(* IEC 61131-3 sources: uPC2_EMCTEST/UPC2_EMCTEST/UPC2_EMCTEST/Source/Definitions, 5 files *)

(* ---- UserDefinedDataType.st.st ---- *)
(*----------------------------------
         ADD HERE YOUR TYPES!
----------------------------------*)
TYPE
    (**STone project GIUD*)
    StonePrjGUID:
        STRUCT
            Grp1 : STRING[8];
            Grp2 : STRING[4];
            Grp3 : STRING[4];
            Grp4 : STRING[4];
            Grp5 : STRING[12];
        END_STRUCT;

    (**Date position range*)
    DatePosRange : UINT(0..99);

    (**Time Struct used to change RTC*)
    TimeRTC: STRUCT
        (**Hourh*)  {ATTRIBUTE UOM HOUR}
        Hour        : UINT(0..23);
        (**Minute*) {ATTRIBUTE UOM MINUTE}
        Minute      : UINT(0..59);
        (**Second*){ATTRIBUTE UOM SECOND}
        Second      : UINT(0..59);
        (**Millisecond*){ATTRIBUTE UOM MILLISECOND}
        Millisecond : UINT(0..999);
    END_STRUCT;

    (**Date Struct used to change RTC*)
    DateRTC: STRUCT
        (**Day*)    {ATTRIBUTE UOM DAY}
        Day         : UINT(1..31);
        (**Month*)  {ATTRIBUTE UOM MONTH}
        Month       : UINT(1..12);
        (**Year*)   {ATTRIBUTE UOM YEAR}
        Year        : UINT(2021..2200);
    END_STRUCT;

    (**Date and time Struct used to change RTC*)
    DateTimeRTC: STRUCT
        (**Day*)    {ATTRIBUTE UOM DAY}
        Day         : UINT(1..31);
        (**Month*)  {ATTRIBUTE UOM MONTH}
        Month       : UINT(1..12);
        (**Year*)   {ATTRIBUTE UOM YEAR}
        Year        : UINT(2021..2200);
        (**Hourh*)  {ATTRIBUTE UOM HOUR}
        Hour        : UINT(0..23);
        (**Minute*) {ATTRIBUTE UOM MINUTE}
        Minute      : UINT(0..59);
        (**Second*){ATTRIBUTE UOM SECOND}
        Second      : UINT(0..59);
        (**Millisecond*){ATTRIBUTE UOM MILLISECOND}
        Millisecond : UINT(0..999);
    END_STRUCT;

    (**Units measure zone*)
    UOM_ZONE :
        (
        (**No Zone*)
        NONE,
        (**International System Zone [°C/bar]*)
        SI,
        (**Imperial Zone [°F/psi]*)
        Imperial
        );

   (**Unit status type*)
    UNIT_STATUS:
    (
        NOT_Used,                   (**Bacnet compatibility*)
        UnitON,                     (**Unit ON*)
        OffByAlarm,                 (**Off By Alarm*)
        OffByBMS,                   (**Off By BMS*)
        OffByScheduler,             (**Off By Scheduler*)
        OffByDI,                    (**Off By Digital Input*)
        OffByKeyboard,              (**Off By Keyboard*)
        OffByNetwork,               (**Off By Network*)
        Manual,                     (**Unit manual mode active*)
        ChangeOver,                 (**ChangeOver*)
        SwitchON,                   (**Switch ON*)
        ShutDown,                   (**Shut Down*)
        PreConditioning,            (**Pre-Conditioning*)
        Dehumidification,           (**Dehumidification*)
        Antifreeze,                 (**Antifreeze*)
        Defrost,                    (**Defrost*)
        AirPressure_Flow,           (**Air Pressure/Flow*)
        AirQuality,                 (**Air Quality*)
        Cooling,                    (**Cooling*)
        Heating,                    (**Heating*)
        FreeCooling,                (**FreeCooling*)
        FreeHeating,                (**FreeHeating*)
        LowTemperatureControl,      (**Low Temperature Control*)
        HighTemperatureControl,     (**High Temperature Control*)
        TestIO,                     (**Test I/O*)
        DHW,                        (**Domestic Hot Water*)
        InactivityStart,            (**Inactivity Start*)
        HighSaturationHumidity,     (**High Saturation Humidity*)
        Purging                     (**Purging*)
    );

    (**List of Quick Menu position*)
    QUICK_MENU:
    (
        (**Selected Loop OnOff*)
        OnOff,
        (**Selcted Loop Set*)
        Set,
        (**Selected Loop Info*)
        Info
    );

    (**Current state of HMI - Used to manage LogoMask/LanguageMask/MainMask transition*)
    State_HMI:
    (
        Wait,
        DisplayLogoMask,
        DisplayLanguageMask,
        DisplayMainMask
    );

    (**Serial port configuration (Parity and Stop bits)*)
    Serial_ParityStopBits :
    (
        (**NONE-1*)
        NONE_1,
        (**NONE-2*)
        NONE_2,
        (**EVEN-1*)
        EVEN_1,
        (**EVEN-2*)
        EVEN_2,
        (**ODD-1*)
        ODD_1,
        (**ODD-2*)
        ODD_2
    );

    (**Serial port baud rate configuration*)
    Serial_Speed :
    (
        (**Baud rate 1200*)
        Baud_1200,
        (**Baud rate 2400*)
        Baud_2400,
        (**Baud rate 4800*)
        Baud_4800,
        (**Baud rate 9600*)
        Baud_9600,
        (**Baud rate 19200*)
        Baud_19200,
        (**Baud rate 38400*)
        Baud_38400,
        (**Baud rate 57600*)
        Baud_57600,
        (**Baud rate 115200*)
        Baud_115200,
        (**Baud rate 375000*)
        Baud_375000
    );

    (**Type of password used for Login procedure*)
    LOGIN_PASSWORD :
    (
        User,
        Service,
        Manufacturer,
        System
    );

    (**Used by APPLICA to manage clock and timezone*)
    APPsConfigRTC:
        STRUCT
        	(**Every time it's value change the PLC change it's RTC*)
        	SetRTC     : BOOL;
            (**New "Date and Time" used to update the RTC*)
        	DateTime   : DATE_AND_TIME;
        	(**New "Time Zone" used to update the RTC*)
        	TimeZone   : STRING;
        END_STRUCT;

END_TYPE

(* ---- VAR_GLOBAL.st ---- *)
USING System;
USING System.Timer;
(*----------------------------------
         ADD HERE YOUR VARS!
----------------------------------*)
VAR_GLOBAL
    (**Restore application to defualt settings (FALSE=Disabled, TRUE=Enabled)*)
	Restoredefault   : BOOL;
    (**Instance to manage comunication between Client&Salve in Modbus client protocol with Fieldbus port*)
//    ClientModbus_pCO : MBM_Template_pCO;

    {REGION SYSTEM INFO}
        (**Retain writings number*)
        RetainWrN       : UDINT;
        (**Task Main live counter*)
        TaskMainLiveCnt : UINT;
        (**Task Main execution time*)
        {ATTRIBUTE UOM MILLISECOND}
        TaskMainExeT    : UDINT;
        (**Current System Time*)
        {ATTRIBUTE UOM MILLISECOND}
        CurrSysT        : UDINT;
        (**Task Main current execution time*)
        {ATTRIBUTE UOM MILLISECOND}
        TaskMainCurrT   : UDINT;

        (**System Info structure*)
        SysInfo         : SystemInfo;
        (**Hardware Info structure*)
        HardwareInfo    : HardwareDescription;
        (**Prject information*)
        InfoProject     : ProjectInfo;
        (**Product information read in OTP memory*)
        InfoProduct     : ProductInfo;

        (**PLC SW can GO*)
        Go_PLC          : BOOL;

        (**Device model*)
		DeviceType      : UINT;
        (**Board type*)
        BoardType       : UINT;
        (**Target machine type*)
		MachineType     : UINT;
        (**Target hardware code*)
		HwCode          : UINT;

        RetainMemWrites : ULINT;

        (**Stone project GUID*)
        GUID : StonePrjGUID;
    {ENDREGION}

    {REGION Used by APPLICA to manage clock and timeZONE}
        APPsCfgRTC : APPsConfigRTC;
    {ENDREGION}

    {REGION HMI}
        (**Logged in pGD1 display as Service*)
    	Access_Service : BOOL;
        (**Logged in pGD1 display as User*)
    	Access_User    : BOOL;
        (**Logged in pGD1 display as Manufacturer*)
    	Access_Manuf   : BOOL;
        (**Logged in pGD1 display as System Manager*)
    	Access_Sys     : BOOL;
        (**Switch to TRUE or FALSE every second*)
        Blink          : BOOL;
        (**Password used for Loging procedure (User, Service, Manufacturer, System)*) {METADATA MIN_VAL 0} {METADATA MAX_VAL 3}
        LoginPwdType   : USINT;

    	{REGION Management of "Date and Hour" displayed by pGD1 display}
            (**Current local time (read only)*)
            CurrLocTime    : DateTimeRTC;
            (**UTC Date and Time*)
            TimeUTC        : DATE_AND_TIME;
            (**Local Date and Time based on current time zone*)
            LocDateAndTime : DATE_AND_TIME;
            (**Local time based on current time zone*)
            LocTime        : DateTime;
            (**Current day of week*)
            Day_Week       : DayOfWeek(0..6);
            (**Set clock settings by Net*)
            SetClockByNet  : BOOL;
        {ENDREGION}

        {REGION Date and time changing management by Network}
            (**Values of Date and Time used to modify RTC by network*)
            NewDateTimeByNet  : DateTimeRTC;
        {ENDREGION}

        {REGION Date and time changing management by pGD1}
            (**Values of Date and Time used to modify clock by pGD1*)
            DateTimeBypGD1 : TimeRTC;

            (**Date element position P1, the date format is P1/P2/P3*) {METADATA MIN_VAL DateP1Lmin} {METADATA MAX_VAL DateP1Lmax}
            DateP1     : DatePosRange;
            (**Date element position P1 limit min*)
            DateP1Lmin : DatePosRange;
            (**Date element position P1 limit max*)
            DateP1Lmax : DatePosRange;

            (**Date element position P2, the date format is P1/P2/P3*) {METADATA MIN_VAL DateP2Lmin} {METADATA MAX_VAL DateP2Lmax}
            DateP2     : DatePosRange;
            (**Date element position P2 limit min*)
            DateP2Lmin : DatePosRange;
            (**Date element position P2 limit max*)
            DateP2Lmax : DatePosRange;

            (**Date element position P3, the date format is P1/P2/P3*) {METADATA MIN_VAL DateP3Lmin} {METADATA MAX_VAL DateP3Lmax}
            DateP3     : DatePosRange;
            (**Date element position P3 limit min*)
            DateP3Lmin : DatePosRange;
            (**Date element position P3 limit max*)
            DateP3Lmax : DatePosRange;
        {ENDREGION}
    {ENDREGION}

    {REGION ALARMS MANAGEMENT BY HMI}
        (**Some alarms have been triggered by system. It's necessary to reset them*)
	    GblAlarm            : BOOL;
        (**Buzzer status (FALSE=Active, TRUE=Silenced)*)
	    BuzzerSilenced      : BOOL := FALSE;
        (**Requet to make blink LED-Alarm*)
        Req_BlinkLED_Alarm  : BOOL;
        (**Requet to maintain LED-Alarm's light on and fixed)*)
        Req_FixLED_Alarm    : BOOL;
        (**Requet TO make blink LED-PRG*)
        Req_BlinkLED_PRG    : BOOL;
        (**Requet to maintain LED-PRG's light on and fixed)*)
        Req_FixLED_PRG      : BOOL;
    {ENDREGION}

        //New add variable because of buliting error
        MenuWidget1 : MenuWidget;
        SubMenuWidget1 : SubMenuWidget;
        HistoryAlarmsWidget1 : HistoryAlarmsWidget;

    {REGION Management of HMI LEDs}
        (**Mng. of LED blinking Alarm*)
    	DisplayBlinkLED_Alarm      : BOOL;
        (**Mng. of LED Alarm*)
    	DisplayLED_Alarm           : BOOL;
        (**Mng. of LED blinking PRG*)
    	DisplayBlinkLED_PRG        : BOOL;
        (**Mng. of LED PRG*)
    	DisplayLED_PRG             : BOOL;
        (**Mng. of LED blinking BACKGROUND*)
    	DisplayBlinkLED_BACKGROUND : BOOL;
        (**Mng. of LED BACKGROUND*)
        DisplayLED_BACKGROUND      : BOOL;
    {ENDREGION}

    {REGION Unit management}
        (**Unit ON/OFF status (FALSE=ON, TRUE=OFF)*)
    	UnitOff         : BOOL;
    	(**Unit ON/OFF status (FALSE=OFF, TRUE=ON)*)
    	UnitOn          : BOOL;
        (**Unit ON/OFF command by Scheduler (FALSE=On, TRUE=Off)*)
    	SchedOnOff      : BOOL;
    {ENDREGION}

    {REGION Main Mask}
    	(**UnitStatus - Unit status*)
    	UnitStatus      : UNIT_STATUS (UNIT_STATUS#NOT_Used..UNIT_STATUS#Purging);
        (**Index of the Quick Menu*)
        IdxQM           : QUICK_MENU (QUICK_MENU#OnOff..QUICK_MENU#Info);
        (**Index of the image displayed by Quick Menu*)
        IdxImgQM        : USINT (0..5);
    {ENDREGION}

    {REGION Managemnet of Password in pGD1 interface}
        (**Temporary password*)
    	TmpPwd      : UINT(0..9999) := 0;
    	(**Temporary password digit 1*)
    	TmpPwd_Dig1 : UINT(0..9) := 0;
    	(**Temporary password digit 2*)
    	TmpPwd_Dig2 : UINT(0..9) := 0;
    	(**Temporary password digit 3*)
    	TmpPwd_Dig3 : UINT(0..9) := 0;
    	(**Temporary password digit 4*)
    	TmpPwd_Dig4 : UINT(0..9) := 0;
    {ENDREGION}

    {REGION LANGUAGE MASK MANAGEMENT}
        (**Language string displayed inside LanguageSelection mask*)
        LangMskStr : STRING;
        (**Language acronym displayed inside LanguageSelection mask*)
        LangMskAcr : STRING;
    {ENDREGION}

    {REGION BMS1 management}
        (**Applies the settings of serial line BMS1 (Auto-Reset excuted by application)*)
        BMS1_ChangeSet   : BOOL := TRUE;
    {ENDREGION}

    {REGION BMS2 management}
        (**Applies the settings of serial line BMS2 (Auto-Reset excuted by application)*)
        BMS2_ChangeSet   : BOOL := TRUE;
        (**BMS2 net online (a client is quering on BMS net this board)*)
    	BMS2_Online      : BOOL;

        {REGION Used to save BMS2 settings}
            BMS2_Addr_SavedRAM : USINT(1..247);
        	BMS2_Baud_SavedRAM : Serial_Speed;
        	BMS2_Conf_SavedRAM : Serial_ParityStopBits;
        {ENDREGION}

    	(**Unit On/Off command by NET (0=OFF, 1=ON)*)
    	NET_OnOff : BOOL;
    {ENDREGION}

    {REGION FIELDBUS1 MANAGEMENT}
        (**Applies the settings of serial line FB1 (Auto-Reset excuted by application)*)
        FB1_ChangeSet : BOOL := TRUE;
    {ENDREGION}

    {REGION FIELDBUS2 MANAGEMENT}
        (**Applies the settings of serial line FB2 (Auto-Reset excuted by application)*)
        FB2_ChangeSet : BOOL := TRUE;
    {ENDREGION}

    {REGION Unit On}
        (**Reset of all hours counter (FALSE=None, TRUE=Reset)*)
        ResTotCnt    : BOOL;
        (**Unit On hours counter*) {ATTRIBUTE UOM HOUR}
        UnitOnHrs    : UDINT;
        (**Unit On reset hour counters*)
    	UnitOnResHrs : BOOL;
    {ENDREGION}

    {REGION BLACKOUT}
        (**Date of the last power off expressed in seconds (Unix Timestamp, seconds from January 1st 1970)*)
        PwrOffDate_NVRAM_BLKO : UDINT;
        (**Duration of the power off in minutes*)   {METADATA MIN_VAL 0} {METADATA MAX_VAL 59} {ATTRIBUTE UOM MINUTE}
        OffMins_BLKO       :UINT;
        (**Duration of the power off in hours*)     {METADATA MIN_VAL 0} {METADATA MAX_VAL 23} {ATTRIBUTE UOM HOUR}
        OffHours_BLKO      :UINT;
        (**Duration of the power off in days*)      {METADATA MIN_VAL 1} {METADATA MAX_VAL 999} {ATTRIBUTE UOM DAY}
        OffDays_BLKO       :UINT;
        (**Last second in which Plc was on*)        {METADATA MIN_VAL 0} {METADATA MAX_VAL 59} {ATTRIBUTE UOM SECOND}
        LastOnSec_BLKO     :UINT;
        (**Last minute in which Plc was on*)        {METADATA MIN_VAL 0} {METADATA MAX_VAL 59} {ATTRIBUTE UOM MINUTE}
        LastOnMin_BLKO     :UINT;
        (**Last hour in which Plc was on*)          {METADATA MIN_VAL 0} {METADATA MAX_VAL 23} {ATTRIBUTE UOM HOUR}
        LastOnHour_BLKO    :UINT;
        (**Last day in which Plc was on*)           {METADATA MIN_VAL 1} {METADATA MAX_VAL 31} {ATTRIBUTE UOM DAY}
        LastOnDay_BLKO     :UINT;
        (**Last month in which Plc was on*)         {METADATA MIN_VAL 1} {METADATA MAX_VAL 12} {ATTRIBUTE UOM MONTH}
        LastOnMonth_BLKO   :UINT;
        (**Last year in which Plc was on*)          {METADATA MIN_VAL 2021} {METADATA MAX_VAL 2200} {ATTRIBUTE UOM YEAR}
        LastOnYear_BLKO    :UINT;
    {ENDREGION}

END_VAR

(* ---- VAR_GLOBAL_CONSTANT.st ---- *)
USING System;
(*----------------------------------
         ADD HERE YOUR CONSTANTS!
----------------------------------*)

VAR_GLOBAL CONSTANT
    (**Main Task intervall*)
    MAIN_TASK_INTERVAL    : TIME   := T#300ms;
    (**Hours persistent update rate*) {ATTRIBUTE UOM HOUR}
    HRS_PRST_UPD_RATE     : uint := 3;

    {REGION Project Info}
        (**Project autor*)
        PROJ_AUTHOR           : STRING := __PROJ_AUTHOR__;
        (**Project build date*)
        PROJ_BUILD_DATE       : STRING := __PROJ_BUILD_DATE__;
        (**Project build second*) {ATTRIBUTE UOM SECOND}
        PROJ_BUILD_SECOND     : DINT   := __PROJ_BUILD_SECOND__;
        (**Project build hour*) {ATTRIBUTE UOM HOUR}
        PROJ_BUILD_HOUR       : DINT   := __PROJ_BUILD_HOUR__;
        (**Project build minute*) {ATTRIBUTE UOM MINUTE}
        PROJ_BUILD_MINUTE     : DINT   := __PROJ_BUILD_MINUTE__;
        (**Project build day*) {ATTRIBUTE UOM DAY}
        PROJ_BUILD_DAY        : DINT   := __PROJ_BUILD_DAY__;
        (**Project build month*) {ATTRIBUTE UOM MONTH}
        PROJ_BUILD_MONTH      : DINT   := __PROJ_BUILD_MONTH__;
        (**Project build year*) {ATTRIBUTE UOM YEAR}
        PROJ_BUILD_YEAR       : DINT   := __PROJ_BUILD_YEAR__;
        (**Project name*)
        PROJ_NAME             : STRING := __PROJ_NAME__;
        (**Project vendor*)
        PROJ_VENDOR           : STRING := __PROJ_VENDOR__;
        (**Project version*)
        PROJ_VER              : STRING := __PROJ_VER__;
        (**Project version Build*)
        PROJ_VER_BUILD        : DINT   := __PROJ_VER_BUILD__;
        (**Project version Major*)
        PROJ_VER_MAJOR        : DINT   := __PROJ_VER_MAJOR__;
        (**Project version Minor*)
        PROJ_VER_MINOR        : DINT   := __PROJ_VER_MINOR__;
        //PROJ_VER_TYPE         : CHAR   := __PROJ_VER_TYPE__;
    {ENDREGION}

    {REGION Din/Dout logic}
        (**The digital input logic is for command: variable assumes TRUE when contact is closed*)
        DIN_LOGIC_NO : BOOL  := TRUE;
        (**The digital input logic is for alarm: variable assumes TRUE when contact is opened*)
        DIN_LOGIC_NC : BOOL  := FALSE;
        (**The digital out logic is direct: variable assumes TRUE to close the contact (energizing the relay)*)
        DOUT_LOGIC_NO : BOOL := FALSE;
        (**The digital out logic is reverted: variable assumes TRUE to open the contact (de-energizing the relay)*)
        DOUT_LOGIC_NC : BOOL := TRUE;
    {ENDREGION}

    {REGION Ain probe}
        (**Probes alarm delay*) {ATTRIBUTE UOM SECOND}
        PrbDly     : UDINT(0..99) := 10;
        (**Probe filter: number of samples to be averaged (default = 5)*)
        PRB_FILTER : USINT := 5;
    {ENDREGION}

    {REGION TIMEZONE}
    (* TO DELETE! when OS gives API to manage TIME-ZONE*)
        TzIdMax : UINT := 136;
        (**Name of time zone to display in mask*)
        TimeZoneName : ARRAY [1..TzIdMax] OF STRING :=
                                                [
                                                '(UTC-12:00) International Date Line West',
                                                '(UTC-11:00) Coordinated Universal Time-11',
                                                '(UTC-10:00) Aleutian Islands',
                                                '(UTC-10:00) Hawaii',
                                                '(UTC-09:30) Marquesas Islands',
                                                '(UTC-09:00) Alaska',
                                                '(UTC-09:00) Coordinated Universal Time-09',
                                                '(UTC-08:00) Baja California (+others equivalent)',
                                                '(UTC-08:00) Coordinated Universal Time-08',
                                                '(UTC-08:00) Pacific Time (US & Canada)',
                                                '(UTC-07:00) Arizona',
                                                '(UTC-07:00) Chihuahua, La Paz, Mazatlan',
                                                '(UTC-07:00) Mountain Time (US & Canada)',
                                                '(UTC-06:00) Central America (+others equivalent)',
                                                '(UTC-06:00) Central Time (US & Canada)',
                                                '(UTC-06:00) Easter Island',
                                                '(UTC-06:00) Guadalajara, Mexico City, Monterrey',
                                                '(UTC-06:00) Saskatchewan',
                                                '(UTC-05:00) Bogota, Lima, Quito, Rio Branco',
                                                '(UTC-05:00) Chetumal',
                                                '(UTC-05:00) Eastern Time (US & Canada) (+others equivalent)',
                                                '(UTC-05:00) Haiti',
                                                '(UTC-05:00) Havana',
                                                '(UTC-05:00) Indiana (East)',
                                                '(UTC-04:00) Asuncion',
                                                '(UTC-04:00) Atlantic Time (Canada)',
                                                '(UTC-04:00) Caracas (+others equivalent)',
                                                '(UTC-04:00) Cuiaba',
                                                '(UTC-04:00) Georgetown, La Paz, Manaus, San Juan',
                                                '(UTC-04:00) Santiago',
                                                '(UTC-04:00) Turks and Caicos',
                                                '(UTC-03:30) Newfoundland',
                                                '(UTC-03:00) Araguaina (+others equivalent)',
                                                '(UTC-03:00) Brasilia',
                                                '(UTC-03:00) Cayenne, Fortaleza',
                                                '(UTC-03:00) City of Buenos Aires',
                                                '(UTC-03:00) Greenland',
                                                '(UTC-03:00) Montevideo',
                                                '(UTC-03:00) Punta Arenas',
                                                '(UTC-03:00) Saint Pierre and Miquelon',
                                                '(UTC-03:00) Salvador',
                                                '(UTC-02:00) Coordinated Universal Time-02 (+others equivalent)',
                                                '(UTC-02:00) Mid-Atlantic - Old',
                                                '(UTC-01:00) Azores',
                                                '(UTC-01:00) Cabo Verde Is.',
                                                '(UTC) Coordinated Universal Time',
                                                '(UTC+00:00) Casablanca',
                                                '(UTC+00:00) Dublin, Edinburgh, Lisbon, London',
                                                '(UTC+00:00) Monrovia, Reykjavik',
                                                '(UTC+01:00) Amsterdam, Berlin, Bern, Rome, Stockholm, Vienna (+others equiv.)',
                                                '(UTC+01:00) Belgrade, Bratislava, Budapest, Ljubljana, Prague',
                                                '(UTC+01:00) Brussels, Copenhagen, Madrid, Paris',
                                                '(UTC+01:00) Sarajevo, Skopje, Warsaw, Zagreb',
                                                '(UTC+01:00) West Central Africa',
                                                '(UTC+01:00) Windhoek (+others equivalent)',
                                                '(UTC+02:00) Amman',
                                                '(UTC+02:00) Athens, Bucharest (+others equivalent)',
                                                '(UTC+02:00) Beirut',
                                                '(UTC+02:00) Cairo (+others equivalent)',
                                                '(UTC+02:00) Chisinau',
                                                '(UTC+02:00) Damascus',
                                                '(UTC+02:00) Gaza, Hebron',
                                                '(UTC+02:00) Harare, Pretoria',
                                                '(UTC+02:00) Helsinki, Kyiv, Riga, Sofia, Tallinn, Vilnius',
                                                '(UTC+02:00) Jerusalem',
                                                '(UTC+02:00) Kaliningrad',
                                                '(UTC+02:00) Khartoum',
                                                '(UTC+02:00) Tripoli',
                                                '(UTC+03:00) Baghdad (+others equivalent)',
                                                '(UTC+03:00) Istanbul',
                                                '(UTC+03:00) Kuwait, Riyadh',
                                                '(UTC+03:00) Minsk',
                                                '(UTC+03:00) Moscow, St. Petersburg, Volgograd',
                                                '(UTC+03:00) Nairobi',
                                                '(UTC+03:30) Tehran',
                                                '(UTC+04:00) Abu Dhabi, Muscat (+others equivalent)',
                                                '(UTC+04:00) Astrakhan, Ulyanovsk',
                                                '(UTC+04:00) Baku',
                                                '(UTC+04:00) Izhevsk, Samara',
                                                '(UTC+04:00) Port Louis',
                                                '(UTC+04:00) Saratov',
                                                '(UTC+04:00) Tbilisi',
                                                '(UTC+04:00) Yerevan',
                                                '(UTC+04:30) Kabul',
                                                '(UTC+05:00) Ashgabat, Tashkent (+others equivalent)',
                                                '(UTC+05:00) Ekaterinburg',
                                                '(UTC+05:00) Islamabad, Karachi',
                                                '(UTC+05:30) Chennai, Kolkata, Mumbai, New Delhi',
                                                '(UTC+05:30) Sri Jayawardenepura',
                                                '(UTC+05:45) Kathmandu',
                                                '(UTC+06:00) Astana (+others equivalent)',
                                                '(UTC+06:00) Dhaka',
                                                '(UTC+06:00) Omsk',
                                                '(UTC+06:30) Yangon (Rangoon)',
                                                '(UTC+07:00) Bangkok, Hanoi, Jakarta (+others equivalent)',
                                                '(UTC+07:00) Barnaul, Gorno-Altaysk',
                                                '(UTC+07:00) Hovd',
                                                '(UTC+07:00) Krasnoyarsk',
                                                '(UTC+07:00) Novosibirsk',
                                                '(UTC+07:00) Tomsk',
                                                '(UTC+08:00) Beijing, Chongqing, Hong Kong, Urumqi (+others equivalent)',
                                                '(UTC+08:00) Irkutsk (+others equivalent)',
                                                '(UTC+08:00) Kuala Lumpur, Singapore',
                                                '(UTC+08:00) Perth',
                                                '(UTC+08:00) Taipei',
                                                '(UTC+08:00) Ulaanbaatar',
                                                '(UTC+08:30) Pyongyang (+others equivalent)',
                                                '(UTC+08:45) Eucla',
                                                '(UTC+09:00) Chita (+others equivalent)',
                                                '(UTC+09:00) Osaka, Sapporo, Tokyo',
                                                '(UTC+09:00) Seoul',
                                                '(UTC+09:00) Yakutsk',
                                                '(UTC+09:30) Adelaide',
                                                '(UTC+09:30) Darwin',
                                                '(UTC+10:00) Brisbane',
                                                '(UTC+10:00) Canberra, Melbourne, Sydney (+others equivalent)',
                                                '(UTC+10:00) Guam, Port Moresby (+others equivalent)',
                                                '(UTC+10:00) Hobart',
                                                '(UTC+10:00) Vladivostok',
                                                '(UTC+10:30) Lord Howe Island',
                                                '(UTC+11:00) Bougainville Island (+others equivalent)',
                                                '(UTC+11:00) Chokurdakh',
                                                '(UTC+11:00) Magadan',
                                                '(UTC+11:00) Norfolk Island',
                                                '(UTC+11:00) Sakhalin',
                                                '(UTC+11:00) Solomon Is., New Caledonia',
                                                '(UTC+12:00) Anadyr, Petropavlovsk-Kamchatsky (+others equivalent)',
                                                '(UTC+12:00) Auckland, Wellington',
                                                '(UTC+12:00) Coordinated Universal Time+12',
                                                '(UTC+12:00) Fiji',
                                                '(UTC+12:00) Petropavlovsk-Kamchatsky - Old',
                                                '(UTC+12:45) Chatham Islands',
                                                '(UTC+13:00) Coordinated Universal Time+13 (+others equivalent)',
                                                '(UTC+13:00) Nuku alofa',
                                                '(UTC+13:00) Samoa',
                                                '(UTC+14:00) Kiritimati Island'
                                            ];
        (**Time zone POSIX rule.*)
        TimeZonePOSIX : ARRAY [1..TzIdMax] OF STRING :=
                                            [
                                            '<-12>12',
                                            '<-11>11',
                                            'HST10HDT,M3.2.0,M11.1.0',
                                            'HST10',
                                            '<-0930>9:30',
                                            'AKST9AKDT,M3.2.0,M11.1.0',
                                            '<-09>9',
                                            'PST8PDT,M3.2.0,M11.1.0',
                                            '<-08>8',
                                            'PST8PDT,M3.2.0,M11.1.0',
                                            'MST7',
                                            'MST7MDT,M4.1.0,M10.5.0',
                                            'MST7MDT,M3.2.0,M11.1.0',
                                            'CST6',
                                            'CST6CDT,M3.2.0,M11.1.0',
                                            '<-06>6<-05>,M9.1.6/22,M4.1.6/22',
                                            'CST6CDT,M4.1.0,M10.5.0',
                                            'CST6',
                                            '<-05>5',
                                            'EST5',
                                            'EST5EDT,M3.2.0,M11.1.0',
                                            'EST5EDT,M3.2.0,M11.1.0',
                                            'CST5CDT,M3.2.0/0,M11.1.0/1',
                                            'EST5EDT,M3.2.0,M11.1.0',
                                            '<-04>4<-03>,M10.1.0/0,M3.4.0/0',
                                            'AST4ADT,M3.2.0,M11.1.0',
                                            '<-04>4',
                                            '<-04>4<-03>,M11.1.0/0,M2.3.0/0',
                                            '<-04>4',
                                            '<-04>4<-03>,M9.1.0/0,M4.1.0/0',
                                            'EST5EDT,M3.2.0,M11.1.0',
                                            'NST3:30NDT,M3.2.0,M11.1.0',
                                            '<-03>3',
                                            '<-03>3<-02>,M11.1.0/0,M2.3.0/0',
                                            '<-03>3',
                                            '<-03>3',
                                            '<-03>3<-02>,M3.5.6/22,M10.5.6/23',
                                            '<-03>3',
                                            '<-03>3',
                                            '<-03>3<-02>,M3.2.0,M11.1.0',
                                            '<-03>3',
                                            '<-02>2',
                                            '<-02>2',
                                            '<-01>1<+00>,M3.5.0/0,M10.5.0/1',
                                            '<-01>1',
                                            'UTC0',
                                            '<+01>-1',
                                            'GMT0BST,M3.5.0/1,M10.5.0',
                                            'GMT0',
                                            'CET-1CEST,M3.5.0,M10.5.0/3',
                                            'CET-1CEST,M3.5.0,M10.5.0/3',
                                            'CET-1CEST,M3.5.0,M10.5.0/3',
                                            'CET-1CEST,M3.5.0,M10.5.0/3',
                                            'WAT-1',
                                            'CAT-2',
                                            'EET-2EEST,M3.4.5/0,M10.5.5/1',
                                            'EET-2EEST,M3.5.0/3,M10.5.0/4',
                                            'EET-2EEST,M3.5.0/0,M10.5.0/0',
                                            'EET-2',
                                            'EET-2EEST,M3.5.0,M10.5.0/3',
                                            'EET-2EEST,M3.5.5/0,M10.5.5/0',
                                            'EET-2EEST,M3.5.6/1,M10.5.6/1',
                                            'SAST-2',
                                            'EET-2EEST,M3.5.0/3,M10.5.0/4',
                                            'IST-2IDT,M3.5.5,M10.5.0',
                                            'EET-2',
                                            'CAT-2',
                                            'EET-2',
                                            '<+03>-3',
                                            '<+03>-3',
                                            '<+03>-3',
                                            '<+03>-3',
                                            'MSK-3',
                                            'EAT-3',
                                            '<+0330>-3:30<+0430>,M3.4.1/0,M9.4.3/0',
                                            '<+04>-4',
                                            '<+04>-4',
                                            '<+04>-4',
                                            '<+04>-4',
                                            '<+04>-4',
                                            '<+04>-4',
                                            '<+04>-4',
                                            '<+04>-4',
                                            '<+0430>-4:30',
                                            '<+05>-5',
                                            '<+05>-5',
                                            'PKT-5',
                                            'IST-5:30',
                                            '<+0530>-5:30',
                                            '<+0545>-5:45',
                                            '<+06>-6',
                                            '<+06>-6',
                                            '<+06>-6',
                                            '<+0630>-6:30',
                                            '<+07>-7',
                                            '<+07>-7',
                                            '<+07>-7',
                                            '<+07>-7',
                                            '<+07>-7',
                                            '<+07>-7',
                                            'CST-8',
                                            '<+08>-8',
                                            '<+08>-8',
                                            'AWST-8',
                                            'CST-8',
                                            '<+08>-8',
                                            'KST-9',
                                            '<+0845>-8:45',
                                            '<+09>-9',
                                            'JST-9',
                                            'KST-9',
                                            '<+09>-9',
                                            'ACST-9:30ACDT,M10.1.0,M4.1.0/3',
                                            'ACST-9:30',
                                            'AEST-10',
                                            'AEST-10AEDT,M10.1.0,M4.1.0/3',
                                            '<+10>-10',
                                            'AEST-10AEDT,M10.1.0,M4.1.0/3',
                                            '<+10>-10',
                                            '<+1030>-10:30<+11>-11,M10.1.0,M4.1.0',
                                            '<+11>-11',
                                            '<+11>-11',
                                            '<+11>-11',
                                            '<+11>-11',
                                            '<+11>-11',
                                            '<+11>-11',
                                            '<+12>-12',
                                            'NZST-12NZDT,M9.4.0,M4.1.0/3',
                                            '<+12>-12',
                                            '<+12>-12<+13>,M11.1.0,M1.3.0/3',
                                            '<+12>-12',
                                            '<+1245>-12:45<+1345>,M9.4.0/2:45,M4.1.0/3:45',
                                            '<+13>-13',
                                            '<+13>-13',
                                            '<+13>-13<+14>,M9.4.0/3,M4.1.0/4',
                                            '<+14>-14'
                                            ];
    {ENDREGION}
END_VAR

(* ---- VAR_GLOBAL_PERSISTENT.st ---- *)
(*----------------------------------
    ADD HERE YOUR VARS!
----------------------------------*)
VAR_GLOBAL PERSISTENT

    {REGION HMI}
        (**Return to main mask after 300 seconds*)
        {ATTRIBUTE UOM SECOND}
        ReturnMainMaskTime : UINT(0..9999) := 300;
        (**Units measure zone used in HMI*)
    	UoMZoneHMI         : UOM_ZONE := UOM_ZONE#SI;
        (**Date format enum. set by DateTimeChg mask (0=DD/MM/YYYY, 1=MM/DD/YYYY, 2=YYYY/MM/DD)*)
        DateFrmt           : DateFormat(DateFormat#DDMMYYYY..DateFormat#YYYYMMDD) := DateFormat#DDMMYYYY;
        (**Timezone*) {METADATA MIN_VAL 1} {METADATA MAX_VAL 136}
        Timezone           : UINT(1..136) := 50;  (*50=ROME and POSIX is 'CET-1CEST,M3.5.0,M10.5.0/3'*)
    {ENDREGION}

    {REGION ALARMS MANAGEMENT BY HMI}
        (**Enable buzzer (FALSE=Disabled, TRUE=Enabled)*)
    	En_Buzzer : BOOL := TRUE;
    {ENDREGION}

    {REGION LANGUAGE MANAGEMENT}
        (**Shows the language mask at the first SW start up to select language*)
        ShowMskLanguage   : BOOL := TRUE;
        (**Save language*)
        LanguageID      : UINT := 2;
    {ENDREGION}

    {REGION LOGIN MANAGEMENT}
        (**System password*)        {METADATA MIN_VAL 0} {METADATA MAX_VAL 9999}
        PwdSys        : UINT (0..9999) := 1604;
        (**User password*)          {METADATA MIN_VAL 0} {METADATA MAX_VAL 9999}
        PwdUser       : UINT (0..9999) := 0000;
        (**Service password*)       {METADATA MIN_VAL 0} {METADATA MAX_VAL 9999}
        PwdService    : UINT (0..9999) := 1234;
        (**Manufacturer password*)  {METADATA MIN_VAL 0} {METADATA MAX_VAL 9999}
        PwdManuf      : UINT (0..9999) := 9999;
    {ENDREGION}

    {REGION Probes settings}
        (**SetP setpoint*)
    	{ATTRIBUTE UOM CELSIUS}
    	{METADATA MIN_VAL 15.0}
    	{METADATA MAX_VAL 25.0}
    	SetT : REAL := 15.0;
    {ENDREGION}

    {REGION BMS1/2 management}
        (**Enable unit ON/OFF command by BMS net (0=Disabled, 1=Enabled)*)
    	En_BmsOffOn : BOOL := FALSE;
        (**Unit On/Off command by BMS (0=OFF, 1=ON)*)
        BmsOffOn    : BOOL := FALSE;
    {ENDREGION}

    {REGION BMS1 settings}
        (**BMS port serial address*)
        {METADATA MIN_VAL 1} {METADATA MAX_VAL 247}
    	BMS1_Addr    : USINT(1..247) := 1;
    	(**BMS port baud rate (0=1200, 1=2400, 2=4800, 3=9600, 4=19200, 5=38400, 6=57600, 7=115200, 8=375000)*)
    	BMS1_Baud    : Serial_Speed (Serial_Speed#Baud_1200..Serial_Speed#Baud_375000):= Serial_Speed#Baud_19200;
    	(**BMS port network settings (0=NONE-1, 1=NONE-2, 2=EVEN-1, 3=EVEN-2, 4=ODD-1, 5=ODD-2)*)
    	BMS1_Conf    : Serial_ParityStopBits (Serial_ParityStopBits#NONE_1..Serial_ParityStopBits#ODD_2) := Serial_ParityStopBits#NONE_2;
    {ENDREGION}

    {REGION BMS2 settings}
        (**BMS2 port serial address*)
        {METADATA MIN_VAL 1} {METADATA MAX_VAL 247}
    	BMS2_Addr    : USINT(1..247) := 1;
    	(**BMS2 port baud rate (0=1200, 1=2400, 2=4800, 3=9600, 4=19200, 5=38400, 6=57600, 7=115200, 8=375000)*)
    	BMS2_Baud    : Serial_Speed (Serial_Speed#Baud_1200..Serial_Speed#Baud_375000):= Serial_Speed#Baud_19200;
    	(**BMS2 port network settings (0=NONE-1, 1=NONE-2, 2=EVEN-1, 3=EVEN-2, 4=ODD-1, 5=ODD-2)*)
    	BMS2_Conf    : Serial_ParityStopBits (Serial_ParityStopBits#NONE_1..Serial_ParityStopBits#ODD_2) := Serial_ParityStopBits#NONE_2;
    {ENDREGION}

    {REGION FIELDBUS1 settings}
	    (**Enable Fieldbus1 protocol (0=Disabled, 1=Enabled)*)
	    En_FB1   : BOOL := FALSE;
    	(**FiledBus1 port baud rate (0=1200, 1=2400, 2=4800, 3=9600, 4=19200, 5=38400, 6=57600, 7=115200, 8=375000)*)
    	FB1_Baud : Serial_Speed (Serial_Speed#Baud_1200..Serial_Speed#Baud_375000):= Serial_Speed#Baud_19200;
    	(**FiledBus1 port network settings (0=NONE-1, 1=NONE-2, 2=EVEN-1, 3=EVEN-2, 4=ODD-1, 5=ODD-2)*)
    	FB1_Conf : Serial_ParityStopBits (Serial_ParityStopBits#NONE_1..Serial_ParityStopBits#ODD_2) := Serial_ParityStopBits#NONE_2;
    {ENDREGION}

    {REGION FIELDBUS2 settings}
	    (**Enable Fieldbus2 protocol (0=Disabled, 1=Enabled)*)
	    En_FB2   : BOOL := FALSE;
    	(**FiledBus2 port baud rate (0=1200, 1=2400, 2=4800, 3=9600, 4=19200, 5=38400, 6=57600, 7=115200, 8=375000)*)
    	FB2_Baud : Serial_Speed (Serial_Speed#Baud_1200..Serial_Speed#Baud_375000):= Serial_Speed#Baud_19200;
    	(**FiledBus2 port network settings (0=NONE-1, 1=NONE-2, 2=EVEN-1, 3=EVEN-2, 4=ODD-1, 5=ODD-2)*)
    	FB2_Conf : Serial_ParityStopBits (Serial_ParityStopBits#NONE_1..Serial_ParityStopBits#ODD_2) := Serial_ParityStopBits#NONE_2;
    {ENDREGION}

    {REGION ALARMS}
        (**U005- Alarm relay configuration (0=Regulation alarms, 1=All alarms)*)
    	AlarmRelayCfg : BOOL := FALSE;
        (**Enable status of remote alarm by Din (FALSE=Disabled, TRUE=Enabled)*)
        En_DinAlrm    : BOOL := FALSE;
    {ENDREGION}

    {REGION Unit On hours counter}
        (**Unit On working hours (partial)*)
    	{ATTRIBUTE UOM HOUR}
    	UnitOnHrsPartial : UDINT;
    	(**Unit On working hours (total)*)
    	{ATTRIBUTE UOM HOUR}
    	UnitOnHrsTot     : UDINT;
    {ENDREGION}

    {REGION On/Off by Din }
        (**Enable On/Off by Din*)
        En_DinOffOn : BOOL := FALSE;
    {ENDREGION}
END_VAR

(* ---- VAR_GLOBAL_RETAIN.st ---- *)
(*----------------------------------
    ADD HERE YOUR RETAIN VARS!
----------------------------------*)

VAR_GLOBAL RETAIN
	(**UnSt - Unit ON/OFF command by keyboard (0=OFF 1=ON)*)
	KeybOnOff                   : BOOL := FALSE;
    (**Debug Force Product Code*)
    Dbg_ForceProductCode        : BOOL;
    (**Debug force BMS2 online*)
    Dbg_BMS2Online               : BOOL;
END_VAR
